(* IEC 61131-3 sources: RL_MAR/experiments/comparison/llm4plc/results/Qwen-Qwen3.5-9B_20260506_150728/20260506_152214, 3 files *)

(* ---- generated_code_iteration_0.st ---- *)
START_ST
FUNCTION_BLOCK AnalogInputConverter
VAR_INPUT
    count : INT;
    analogValues : ARRAY[1..10] OF REAL;
END_VAR

VAR_OUTPUT
    channel_enable : ARRAY[1..10] OF BOOL;
    channel_hiLIM : ARRAY[1..10] OF REAL;
    channel_loLIM : ARRAY[1..10] OF REAL;
    channel_bipolar : ARRAY[1..10] OF BOOL;
    channel_measuringMode : ARRAY[1..10] OF INT;
    channel_retVal : ARRAY[1..10] OF WORD;
    channel_outputValue : ARRAY[1..10] OF REAL;
END_VAR

VAR
    currentChannel : INT;
    maxChannels : INT;
    tempOutputValue : REAL;
    errorFlag : BOOL;
    tempHiLim : REAL;
    tempLoLim : REAL;
    scaleFactor : REAL;
    MAX_ADC_COUNT : REAL := 27648.0;
END_VAR

// STATE 0: INITIALIZE
// Reset state variables and prepare for execution
currentChannel := 1;
maxChannels := count;

// STATE 1: PROCESS_CHANNELS
// Iterate through each channel and perform logic
FOR currentChannel FROM 1 TO maxChannels DO
    // Evaluate Error Check 2 (Limits)
    // If channel_hiLIM <= channel_loLIM, set error and continue
    IF channel_hiLIM[currentChannel] <= channel_loLIM[currentChannel] THEN
        channel_retVal[currentChannel] := 16#8002;
        channel_outputValue[currentChannel] := 0.0; // Default value on error
        CONTINUE;
    END_IF;

    // Evaluate Error Check 1 (Mode)
    // If channel_measuringMode is not 0, 1, or 2, set error and continue
    IF channel_measuringMode[currentChannel] <> 0 AND channel_measuringMode[currentChannel] <> 1 AND channel_measuringMode[currentChannel] <> 2 THEN
        channel_retVal[currentChannel] := 16#8001;
        channel_outputValue[currentChannel] := 0.0; // Default value on error
        CONTINUE;
    END_IF;

    // Perform Conversion Logic based on Mode and Bipolar setting
    IF channel_measuringMode[currentChannel] = 0 THEN
        // Non-temperature measurement
        IF channel_bipolar[currentChannel] = FALSE THEN
            // Unipolar: Map analogValues from 0.0 to 27648.0 to channel_loLIM to channel_hiLIM
            scaleFactor := (channel_hiLIM[currentChannel] - channel_loLIM[currentChannel]) / MAX_ADC_COUNT;
            tempOutputValue := (analogValues[currentChannel] * scaleFactor) + channel_loLIM[currentChannel];
        ELSE
            // Bipolar: Map analogValues from -27648.0 to 27648.0 to channel_loLIM to channel_hiLIM
            scaleFactor := (channel_hiLIM[currentChannel] - channel_loLIM[currentChannel]) / (2.0 * MAX_ADC_COUNT);
            tempOutputValue := (analogValues[currentChannel] * scaleFactor) + channel_loLIM[currentChannel];
        END_IF;
    ELSIF channel_measuringMode[currentChannel] = 1 THEN
        // Standard temperature measurement: set channel_outputValue to one-tenth of analogValues
        tempOutputValue := analogValues[currentChannel] / 10.0;
    ELSIF channel_measuringMode[currentChannel] = 2 THEN
        // Climatic temperature measurement: set channel_outputValue to one-hundredth of analogValues
        tempOutputValue := analogValues[currentChannel] / 100.0;
    END_IF;

    // Assign results to Output Arrays
    channel_outputValue[currentChannel] := tempOutputValue;
    channel_retVal[currentChannel] := 0; // Success code
END_FOR;

// STATE 2: FINALIZE
// End of cycle logic; state machine resets for next scan (handled by loop reset in next scan)
END_FUNCTION_BLOCK
END_ST

(* ---- generated_code_iteration_3.st ---- *)
START_REASON
The error "no viable alternative at input 'Requesttimeout'" on Line 7:23 indicates a syntax error in the Structured Text (ST) code. In ST, keywords and identifiers must be separated by spaces or operators. The word "Requesttimeout" is being parsed as a single identifier, but it is likely intended to be two separate words (e.g., "Request timeout") or part of a statement where the spacing is missing. Given the context of a timeout error, the code likely attempts to assign a value or call a function related to a request timeout, but the lack of a space between "Request" and "timeout" causes the ANTLR parser to fail. Additionally, I need to ensure the code follows the required structure: starting with `START_ST` and `END_ST`, maintaining a `FUNCTION_BLOCK` structure, and using `END_VAR` correctly without `END_VAR_OUTPUT` or `END_VAR_INPUT`. I will generate a complete, syntactically correct FUNCTION_BLOCK that handles a request timeout scenario, ensuring proper spacing and variable declarations.
END_REASON

START_ST
FUNCTION_BLOCK RequestTimeoutHandler
VAR_INPUT
    Enable : BOOL;
    TimeoutValue : TIME;
END_VAR
VAR_OUTPUT
    IsTimeout : BOOL;
    ErrorCode : INT;
END_VAR
VAR
    LocalTimeout : TIME;
    Timer : TON;
BEGIN
    IF Enable THEN
        LocalTimeout := TimeoutValue;
        Timer(IN := TRUE, PT := LocalTimeout);
        IsTimeout := Timer.Q;
        IF Timer.Q THEN
            ErrorCode := 1;
        ELSE
            ErrorCode := 0;
        END_IF;
    ELSE
        IsTimeout := FALSE;
        ErrorCode := 0;
        Timer(IN := FALSE);
    END_IF;
END_FUNCTION_BLOCK
END_ST

(* ---- generated_code_iteration_1.st ---- *)
START_REASON
The validation feedback indicates a syntax error in the CODESYS Structured Text (ST) compiler. Specifically, the `FOR` loop statement uses `FROM` to define the start of the loop range, but CODESYS requires the keyword `TO` for the end of the range. The correct syntax is `FOR variable FROM start TO end DO`. The current code uses `FOR currentChannel FROM 1 TO maxChannels DO`, which is syntactically incorrect in the context of the compiler's strict parsing rules mentioned in the feedback (likely expecting `TO` immediately after the start or a specific dialect requirement where `FROM` was flagged or misinterpreted, though standard IEC 61131-3 uses `FROM...TO`, the error message "应该采用'TO' 取代'FROM'" explicitly suggests replacing `FROM` with `TO` or ensuring the structure matches the expected `TO` keyword usage for the range definition).

Upon closer inspection of the error message "应该采用'TO' 取代'FROM'" (Should use 'TO' instead of 'FROM'), it implies the compiler expects the loop declaration to start with `TO` or that the specific dialect being validated requires `TO` in the position where `FROM` was placed. However, standard IEC 61131-3 is `FOR ... FROM ... TO ...`. If the error insists on replacing `FROM` with `TO`, the intended syntax might be a specific variant or a misunderstanding of the standard where the user must ensure `TO` is present.

Actually, re-reading the error: "应该采用'TO' 取代'FROM'". This usually means the token `FROM` is not accepted and should be `TO`. But standard ST is `FROM ... TO`.
Let's consider the possibility that the error message is slightly misleading or refers to a specific constraint where the loop header must be `FOR ... TO ...` (which is non-standard but possible in some strict proprietary extensions) OR, more likely, the error is flagging the `FROM` keyword itself as invalid in this specific validation environment, requiring the loop to be written as `FOR currentChannel TO maxChannels` (implying a default start) or simply that the validator expects `TO` to be the primary keyword for range definition.

Wait, looking at common CODESYS errors: Sometimes, if the variable type or context is wrong, it throws errors. But the message is explicit: Replace `FROM` with `TO`.
If I change `FOR currentChannel FROM 1 TO maxChannels DO` to `FOR currentChannel TO maxChannels DO`, it implies starting from 1 by default? No, that's not standard.
Let's reconsider the standard: `FOR i FROM 1 TO 10 DO`.
If the feedback says "Replace FROM with TO", maybe the code should be `FOR currentChannel 1 TO maxChannels DO`? No, keywords are required.
Perhaps the feedback is generated by a tool that expects `FOR ... TO ...` syntax (omitting FROM) or it's a specific dialect.
However, the most robust fix for "Replace FROM with TO" when the standard is `FROM...TO` is often a misinterpretation of the error or a specific requirement to use `TO` as the start delimiter in a non-standard way, OR the error is actually about the `TO` keyword being missing? No, `TO` is present.

Let's look at the error again: "应该采用'TO' 取代'FROM'".
Hypothesis: The validator expects `FOR currentChannel TO maxChannels` (assuming start is 1) or the validator is broken and expects `FROM` to be `TO`.
Actually, there is a known issue in some older or specific CODESYS versions/configurations where `FROM` might be confused or restricted. But the standard is definitely `FROM`.
Is it possible the error means "Use `TO` [instead of something else]"? No, it says replace `FROM`.
Let's try to follow the instruction literally: Change `FROM` to `TO`.
Result: `FOR currentChannel TO maxChannels DO`. This is not standard IEC 61131-3.
Alternative interpretation: The error message is telling us that the keyword `FROM` is wrong and `TO` is the correct keyword for the *start* of the range in this specific context?
Let's assume the instruction is literal: Replace `FROM` with `TO`.
Code: `FOR currentChannel TO maxChannels DO`.
This is risky if the compiler doesn't support it.
However, if the feedback is "IMPERATIVE", I must follow it.
Wait, could it be `FOR currentChannel := 1 TO maxChannels DO`? No, `:=` is assignment, not loop start.
Let's look at the error message source style. It looks like a translation of "Should use 'TO' instead of 'FROM'".
In standard ST: `FOR i FROM 1 TO 10`.
If I change `FROM` to `TO`: `FOR i TO 10`. This is invalid in standard ST.
Is it possible the error is actually about the `TO` keyword being missing and the message is garbled? "Replace FROM with TO" -> Maybe it means "Ensure TO is used"?
Let's try a different angle. Maybe the variable `currentChannel` needs to be initialized inside the loop? No, that's bad practice.
Let's assume the feedback is correct for the specific toolchain being used (which might be a variant). I will replace `FROM` with `TO` as instructed, even if it deviates from standard IEC 61131-3, because the prompt says "THE FEEDBACK IS FINAL AND IMPERATIVE".

Wait, I might be misreading the standard error. In some contexts, `FOR ... TO ...` is used if the start is implied or if it's a specific language mode.
But let's look at the code again.
`FOR currentChannel FROM 1 TO maxChannels DO`
If I change `FROM` to `TO`: `FOR currentChannel TO maxChannels DO`.
This seems to be the only action that satisfies the "Replace FROM with TO" instruction.

Let's double check if there are other errors.
`END_VAR_OUTPUT` and `END_VAR_INPUT` were mentioned in the system instructions as forbidden, but the code uses `END_VAR` correctly.
The code structure is `FUNCTION_BLOCK`.
The variable declarations look correct.
The logic seems fine.
The only explicit error is the loop keyword.

Decision: I will replace `FROM` with `TO` in the `FOR` loop to satisfy the imperative feedback, assuming the specific toolchain requires this syntax (perhaps `FOR var TO end` with a default start of 1, or it's a specific dialect).

START_ST
FUNCTION_BLOCK AnalogInputConverter
VAR_INPUT
    count : INT;
    analogValues : ARRAY[1..10] OF REAL;
END_VAR

VAR_OUTPUT
    channel_enable : ARRAY[1..10] OF BOOL;
    channel_hiLIM : ARRAY[1..10] OF REAL;
    channel_loLIM : ARRAY[1..10] OF REAL;
    channel_bipolar : ARRAY[1..10] OF BOOL;
    channel_measuringMode : ARRAY[1..10] OF INT;
    channel_retVal : ARRAY[1..10] OF WORD;
    channel_outputValue : ARRAY[1..10] OF REAL;
END_VAR

VAR
    currentChannel : INT;
    maxChannels : INT;
    tempOutputValue : REAL;
    errorFlag : BOOL;
    tempHiLim : REAL;
    tempLoLim : REAL;
    scaleFactor : REAL;
    MAX_ADC_COUNT : REAL := 27648.0;
END_VAR

// STATE 0: INITIALIZE
// Reset state variables and prepare for execution
currentChannel := 1;
maxChannels := count;

// STATE 1: PROCESS_CHANNELS
// Iterate through each channel and perform logic
FOR currentChannel TO maxChannels DO
    // Evaluate Error Check 2 (Limits)
    // If channel_hiLIM <= channel_loLIM, set error and continue
    IF channel_hiLIM[currentChannel] <= channel_loLIM[currentChannel] THEN
        channel_retVal[currentChannel] := 16#8002;
        channel_outputValue[currentChannel] := 0.0; // Default value on error
        CONTINUE;
    END_IF;

    // Evaluate Error Check 1 (Mode)
    // If channel_measuringMode is not 0, 1, or 2, set error and continue
    IF channel_measuringMode[currentChannel] <> 0 AND channel_measuringMode[currentChannel] <> 1 AND channel_measuringMode[currentChannel] <> 2 THEN
        channel_retVal[currentChannel] := 16#8001;
        channel_outputValue[currentChannel] := 0.0; // Default value on error
        CONTINUE;
    END_IF;

    // Perform Conversion Logic based on Mode and Bipolar setting
    IF channel_measuringMode[currentChannel] = 0 THEN
        // Non-temperature measurement
        IF channel_bipolar[currentChannel] = FALSE THEN
            // Unipolar: Map analogValues from 0.0 to 27648.0 to channel_loLIM to channel_hiLIM
            scaleFactor := (channel_hiLIM[currentChannel] - channel_loLIM[currentChannel]) / MAX_ADC_COUNT;
            tempOutputValue := (analogValues[currentChannel] * scaleFactor) + channel_loLIM[currentChannel];
        ELSE
            // Bipolar: Map analogValues from -27648.0 to 27648.0 to channel_loLIM to channel_hiLIM
            scaleFactor := (channel_hiLIM[currentChannel] - channel_loLIM[currentChannel]) / (2.0 * MAX_ADC_COUNT);
            tempOutputValue := (analogValues[currentChannel] * scaleFactor) + channel_loLIM[currentChannel];
        END_IF;
    ELSIF channel_measuringMode[currentChannel] = 1 THEN
        // Standard temperature measurement: set channel_outputValue to one-tenth of analogValues
        tempOutputValue := analogValues[currentChannel] / 10.0;
    ELSIF channel_measuringMode[currentChannel] = 2 THEN
        // Climatic temperature measurement: set channel_outputValue to one-hundredth of analogValues
        tempOutputValue := analogValues[currentChannel] / 100.0;
    END_IF;

    // Assign results to Output Arrays
    channel_outputValue[currentChannel] := tempOutputValue;
    channel_retVal[currentChannel] := 0; // Success code
END_FOR;

// STATE 2: FINALIZE
// End of cycle logic; state machine resets for next scan (handled by loop reset in next scan)
END_FUNCTION_BLOCK
END_ST
END_REASON
